(* PLC project Unnamed, Unknown Unnamed 1 *)
(* stored: creationDateTime 2026-05-07T11:47:46, modificationDateTime 2026-05-07T11:47:46 *)

PROGRAM main
  VAR
    Timer_Pause : TON;
    Timer_Lys : TON;
    TimerLysOn : BOOL;
    PresetTime : TIME := T#600ms;
    PresetTime1 : TIME := T#300ms;
    REDLed : BOOL;
  END_VAR

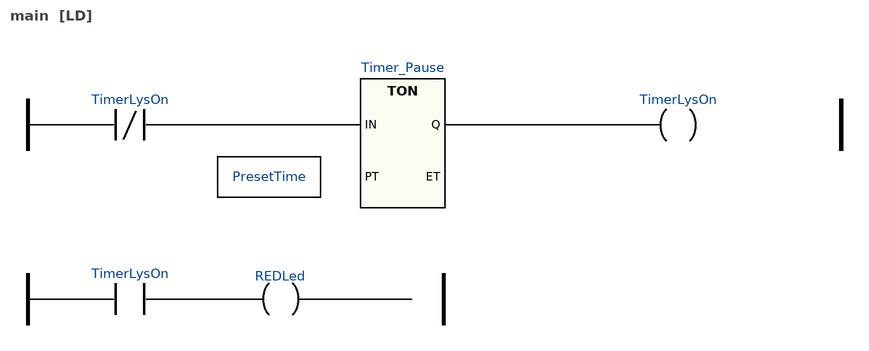
(* LD diagram, written out as Structured Text *)
Timer_Pause(IN := NOT TimerLysOn, PT := PresetTime);
TimerLysOn := Timer_Pause.Q;
REDLed := TimerLysOn;
END_PROGRAM

CONFIGURATION Config0
  RESOURCE Res0 ON PLC
    TASK task0(INTERVAL := T#50ms, PRIORITY := 1);
    PROGRAM instance0 WITH task0 : main;
  END_RESOURCE
END_CONFIGURATION
